FUNCTION_BLOCK TestEvent EXTENDS TcUnit.FB_TestSuite
VAR_INPUT
END_VAR
VAR_OUTPUT
END_VAR
VAR
END_VAR

create_event();
after_initialisation_alarm_is_not_raised();
after_raising_an_alarm_the_alarm_is_raised();
clear_alarm();
add_multiple_events();
raise_and_clear_multiple_alarms();

METHOD add_multiple_events
VAR_INST
  sut: MultipleEventTestsystem;
END_VAR
TEST('Add multiple events');

sut.event1.alarm();
sut.event2.warning();
sut.event3.alarm();
AssertTrue(sut.event1.alarm_raised, 'Event 1');
AssertFalse(sut.event2.alarm_raised, 'Event 2');
AssertTrue(sut.event3.alarm_raised, 'Event 3');

TEST_FINISHED();
END_METHOD

METHOD after_initialisation_alarm_is_not_raised
VAR_INPUT
END_VAR
VAR_INST
  sut: EventTestsystem;
END_VAR
TEST('Alarm is not raised after initialisation');

AssertFalse(sut.event.alarm_raised, '');

TEST_FINISHED();
END_METHOD

METHOD after_raising_an_alarm_the_alarm_is_raised
VAR_INPUT
END_VAR
VAR_INST
  sut: EventTestsystem;
END_VAR
TEST('After raising an alarm the alarm is raised');

sut.event.alarm();
AssertTrue(sut.event.alarm_raised, '');

TEST_FINISHED();
END_METHOD

METHOD clear_alarm
VAR_INPUT
END_VAR
VAR_INST
  sut: EventTestsystem;
END_VAR
TEST('Clear alarm');

sut.event.alarm();
sut.event.clear_alarm();
AssertFalse(sut.event.alarm_raised, '');

TEST_FINISHED();
END_METHOD

METHOD create_event
VAR_INPUT
END_VAR
VAR_INST
  sut: EventTestsystem;
END_VAR
TEST('Create event');

sut.event.message := 'Test';
AssertEquals_STRING('Test', sut.event.message, 'Event not properly created');

TEST_FINISHED();
END_METHOD

METHOD raise_and_clear_multiple_alarms
VAR_INST
  sut: MultipleEventTestsystem;
END_VAR
TEST('Raise and clear multiple alarms');

sut.event1.alarm();
sut.event2.alarm();
sut.event3.alarm();
sut.event1.clear_alarm();
sut.event3.clear_alarm();
AssertFalse(sut.event1.alarm_raised, 'Event 1');
AssertTrue(sut.event2.alarm_raised, 'Event 2');
AssertFalse(sut.event3.alarm_raised, 'Event 3');

TEST_FINISHED();
END_METHOD

END_FUNCTION_BLOCK

(* stored: Version 1.1.0.1, ProductVersion 3.1.4024.9
   POU TestEvent: Id {1f6f0448-1ae3-4068-b11e-400de0fbbc2c}, SpecialFunc None
   Method add_multiple_events: Id {e9dc6e7f-11a1-4018-94b6-f52294564527}
   Method after_initialisation_alarm_is_not_raised: Id {a58568b8-cfac-4930-b4ec-3c7531d956e8}
   Method after_raising_an_alarm_the_alarm_is_raised: Id {3e51c88a-603f-40de-b89e-e09310467482}
   Method clear_alarm: Id {79efaec0-0122-48a3-8419-dd3612e1e2ef}
   Method create_event: Id {84e9d7a6-3a39-48d5-8e25-b4781b9bf70a}
   Method raise_and_clear_multiple_alarms: Id {4d33586e-30c3-471a-bafb-f5eff5aeaf1c} *)
